// TwinCAT 3 PLC project keras2PLC
// ProgramVersion: 3.1.4024.0
// libraries:
//   Real-Time Neural Network generator, * (ISW)
//   Tc2_Standard, * (Beckhoff Automation GmbH)
//   Tc2_System, * (Beckhoff Automation GmbH)
//   Tc2_Utilities, * (Beckhoff Automation GmbH)
//   Tc3_Module, * (Beckhoff Automation GmbH)
// project tree:
//   DUTs/ Dense_v1_Layers.TcDUT, Dense_v1_LayerWeights.TcDUT
//   / PlcTask.TcTTO
//   POUs/achiv/ FB_Dense_v1_load_arch.TcPOU (not stored), FB_Dense_v1_archiv.TcPOU (not stored), MAIN_load_arch.TcPOU (not stored), MAIN_exe_arch.TcPOU
//   POUs/ FB_Dense_v1.TcPOU, MAIN.TcPOU
// real-time tasks:
//   TASK PlcTask: cycle T#10ms, priority 20, ADS port 350

CONFIGURATION keras2PLC
    RESOURCE PLC ON TwinCAT3
        TASK PlcTask(INTERVAL := T#10ms, PRIORITY := 20);
        PROGRAM MAIN WITH PlcTask : MAIN;
    END_RESOURCE
END_CONFIGURATION

// ---- DUTs/Dense_v1_Layers.TcDUT
TYPE Dense_v1_Layers:
STRUCT
    num_layers : UINT := 6;
    weights : Dense_v1_LayerWeights;
    layers : ARRAY[0..5] OF Layer :=[
    (num_neurons := 5),
    (num_neurons := 500, activation := act_type.sigmoid, pointer_weight:= ADR(weights.HiddenLayers1_weight),pointer_bias:= ADR(weights.HiddenLayers1_bias)),
    (num_neurons := 500, activation := act_type.sigmoid, pointer_weight:= ADR(weights.HiddenLayers2_weight),pointer_bias:= ADR(weights.HiddenLayers2_bias)),
    (num_neurons := 500, activation := act_type.sigmoid, pointer_weight:= ADR(weights.HiddenLayers3_weight),pointer_bias:= ADR(weights.HiddenLayers3_bias)),
    (num_neurons := 500, activation := act_type.sigmoid, pointer_weight:= ADR(weights.HiddenLayers4_weight),pointer_bias:= ADR(weights.HiddenLayers4_bias)),
    (num_neurons := 1,activation := act_type.linear,  pointer_weight:= ADR(weights.OutputLayer_weight),pointer_bias:= ADR(weights.OutputLayer_bias))];
    layer_output : ARRAY[0..499] OF LREAL;
    layer_input : ARRAY[0..499] OF LREAL;
    
END_STRUCT
END_TYPE

// ---- DUTs/Dense_v1_LayerWeights.TcDUT
TYPE Dense_v1_LayerWeights:
STRUCT
    normalization_mean : ARRAY[0..0] OF LREAL;
    normalization_std : ARRAY[0..0] OF LREAL;
    HiddenLayers1_weight : ARRAY[0..499,0..4] OF LREAL;
    HiddenLayers1_bias : ARRAY[0..499] OF LREAL;
    HiddenLayers2_weight : ARRAY[0..499,0..499] OF LREAL;
    HiddenLayers2_bias : ARRAY[0..499] OF LREAL;
    HiddenLayers3_weight : ARRAY[0..499,0..499] OF LREAL;
    HiddenLayers3_bias : ARRAY[0..499] OF LREAL;
    HiddenLayers4_weight : ARRAY[0..499,0..499] OF LREAL;
    HiddenLayers4_bias : ARRAY[0..499] OF LREAL;
    OutputLayer_weight : ARRAY[0..0,0..499] OF LREAL;
    OutputLayer_bias : ARRAY[0..0] OF LREAL;
    denormalization_mean : ARRAY[0..0] OF LREAL;
    denormalization_std : ARRAY[0..0] OF LREAL;
    hash_sha_256 : ARRAY[0..3] OF LREAL;
END_STRUCT
END_TYPE

// ---- POUs/MAIN.TcPOU
PROGRAM MAIN
VAR
	vector_2 : ARRAY[0..4] OF LREAL := [1,1,1,1,1];	
	out : ARRAY[0..0] OF LREAL;
	FB_NN : FB_Dense_v1;
	
	runtime_profiler : PROFILER;
	profiler_data : PROFILERSTRUCT;
	
	buf_idx : UINT := 0;
	profiler_buffer : ARRAY [0..1000] OF DWORD;
	
	MeasureFinished : BOOL := TRUE;

	

END_VAR


runtime_profiler(START := TRUE, RESET := TRUE);
FB_NN(pointer_input := ADR(vector_2),pointer_output:= ADR(out));

runtime_profiler(START := FALSE);
profiler_data := runtime_profiler.DATA;
IF NOT MeasureFinished THEN
	profiler_buffer[buf_idx] := profiler_data.LastExecTime;
	buf_idx := buf_idx+1; 
	buf_idx := buf_idx MOD (SIZEOF(profiler_buffer)/SIZEOF(DWORD)); // len of profiler_buffer
	IF buf_idx = 0 THEN
		MeasureFinished := TRUE;
	END_IF
END_IF


//sum := F_DATA_TO_CRC16_CCITT(pData := ADR(FB_NN.nn.weights),cbData := SIZEOF(FB_NN.nn.weights),crc:=crc);
//sum2 := F_CheckSum16(dwSrcAddr := ADR(FB_NN.nn.weights),cbLen := SIZEOF(FB_NN.nn.weights),wChkSum:=crc);

END_PROGRAM

// ---- POUs/FB_Dense_v1.TcPOU
FUNCTION_BLOCK FB_Dense_v1
VAR_INPUT
	pointer_input: POINTER TO LREAL;
	pointer_output : POINTER TO LREAL;
	
END_VAR
VAR	
  i : UINT;
  id : UINT;
  iq : UINT;
  flag_LoadWeights : BOOL := FALSE;
  flag_checkWeights : BOOL := FALSE;
  load_weights : FB_LoadWeights;
  filePath : T_MaxString := 'c:\Users\Administrator\Documents\git-projekte\keras2plc\tests\test_ST_files\Dense_v1_weights.dat';
  nn : Dense_v1_Layers;
  hash_sha_256_twincat : ARRAY[0..3] OF LREAL;
  compare_res : DINT := 99;
  readlen : UINT := 0;
END_VAR

IF NOT flag_LoadWeights THEN
		load_weights(execute := TRUE,filePath := filePath,ReadAdr := ADR(nn.weights), ReadLen :=  readlen);
		IF NOT load_weights.busy THEN 
			flag_LoadWeights := TRUE;
		END_IF
//ELSIF NOT flag_checkWeights THEN
//	F_GenerateHashValue(hashMode:=E_HashMode.HASH_SHA256,pData := ADR(nn.weights),nData := SIZEOF(nn.weights)-32,pHash := ADR(hash_sha_256_twincat),nHash:=32);
//	compare_res := MEMCMp(pBuf1 := ADR(hash_sha_256_twincat),ADR(nn.weights.hash_sha_256),32);
//	IF compare_res = 0 THEN
//		flag_checkWeights := TRUE;
//	END_IF
ELSE
	MEMCPY(destAddr:=ADR(nn.layer_input),srcAddr:=pointer_input,n:=SIZEOF(LREAL)*nn.layers[0].num_neurons);
  // input normalization
	IF nn.layers[0].normalization = act_type.normalization THEN
		FOR id := 0 TO nn.layers[0].num_neurons-1 DO
			 nn.layer_input[id] := F_normalization(x:=nn.layer_input[id],mean:=nn.weights.normalization_mean[id],std:=nn.weights.normalization_std[id]);
	 	END_FOR
	END_IF
  // forward inference
	FOR i := 0 TO nn.num_layers-2 DO
		F_ForwardPropagation(	layer_pre	:= 	nn.layers[i],
								layer_next	:=	nn.layers[i+1],
								pointer_in 	:=	ADR(nn.layer_input),
								pointer_out	:=	ADR(nn.layer_output)	);
		MEMCPY(destAddr:=ADR(nn.layer_input),srcAddr:=ADR(nn.layer_output),n:=SIZEOF(LREAL)*nn.layers[i+1].num_neurons);
	END_FOR
	MEMCPY(destAddr:=pointer_output,srcAddr:=ADR(nn.layer_output),n:=SIZEOF(LREAL)*nn.layers[SIZEOF(nn.layers)/SIZEOF(nn.layers[0])-1].num_neurons);
  // output denormalization
	IF nn.layers[SIZEOF(nn.layers)/SIZEOF(nn.layers[0])-1].normalization = act_type.denormalization THEN
		FOR iq := 0 TO nn.layers[SIZEOF(nn.layers)/SIZEOF(nn.layers[0])-1].num_neurons-1 DO
			 pointer_output[iq] := F_denormalization(x:=pointer_output[iq],mean:=nn.weights.denormalization_mean[iq],std:=nn.weights.denormalization_std[iq]);
	 	END_FOR
	 END_IF
END_IF

END_FUNCTION_BLOCK

// ---- POUs/achiv/MAIN_exe_arch.TcPOU
PROGRAM MAIN_exe_arch
VAR
	vector_2 : ARRAY[0..4] OF LREAL := [1,1,1,1,1];	
	out : ARRAY[0..0] OF LREAL;
	FB_NN : FB_Dense_v1;
	
	runtime_profiler : PROFILER;
	profiler_data : PROFILERSTRUCT;
	
	buf_idx : UINT := 0;
	profiler_buffer : ARRAY [0..1000] OF DWORD;
	
	MeasureFinished : BOOL := True;

END_VAR


runtime_profiler(START := TRUE, RESET := TRUE);
FB_NN(pointer_input := ADR(vector_2),pointer_output:= ADR(out));

runtime_profiler(START := FALSE);
profiler_data := runtime_profiler.DATA;
IF NOT MeasureFinished THEN
	profiler_buffer[buf_idx] := profiler_data.LastExecTime;
	buf_idx := buf_idx+1; 
	buf_idx := buf_idx MOD (SIZEOF(profiler_buffer)/SIZEOF(DWORD)); // len of profiler_buffer
	IF buf_idx = 0 THEN
		MeasureFinished := TRUE;
	END_IF
END_IF


//sum := F_DATA_TO_CRC16_CCITT(pData := ADR(FB_NN.nn.weights),cbData := SIZEOF(FB_NN.nn.weights),crc:=crc);
//sum2 := F_CheckSum16(dwSrcAddr := ADR(FB_NN.nn.weights),cbLen := SIZEOF(FB_NN.nn.weights),wChkSum:=crc);

END_PROGRAM
